// TIA Portal project "OPCUATST" (V15)

(* hardware
DEVICE "S71500/ET200MP station_1"  S7-1500 station
   slot 0: "导轨_0"  Rack  6ES7 590-1***0-0AA0
   slot 1: "PLC_1"  CPU 1515-2 PN  6ES7 515-2AM01-0AB0  V2.5
      slot 3: "CPU 显示_1"  6ES7591-1BA00-0AA0
*)

// ===== PLC "PLC_1"  CPU 1515-2 PN =====

VAR_GLOBAL   // PLC tag table "默认变量表"
   "OPCUATESTBOOL" AT %M0.0 : Bool;
   "OPCUATESTMW" AT %MW1 : Word;
   "OPCUATESTMD" AT %MD4 : DWord;
END_VAR

DATA_BLOCK "DataStatic"   // DB2
{ S7_Optimized_Access := 'TRUE' }
VERSION : 0.1
   VAR
      myBool : Bool := true;
      myByte : Byte := 16#AB;
      myWord : Word := 16#CDEF;
      myDword : DWord := 16#1234567F;
      myInt : Int := 42;
      myUInt : UInt := 65535;
      myString : String := 'Hello World';
      myReal : Real := 9.81;
      myArrayByte : Array[0..127] of Byte;
      myArrayInt : Array[0..127] of Int;
      myArrayUInt : Array[0..127] of UInt;
      myArrayLInt : Array[0..127] of LInt;
      myArrayReal : Array[0..127] of Real;
      myArrayLReal : Array[0..127] of LReal;
      myArrayBool : Array[0..127] of Bool;
   END_VAR
BEGIN
   myArrayByte[0] := 1;
   myArrayByte[1] := 2;
   myArrayByte[2] := 3;
   myArrayByte[3] := 4;
   myArrayByte[4] := 5;
   myArrayByte[5] := 6;
   myArrayByte[6] := 7;
   myArrayByte[7] := 8;
   myArrayByte[8] := 9;
   myArrayByte[9] := 10;
   myArrayByte[10] := 11;
   myArrayByte[11] := 12;
   myArrayByte[12] := 13;
   myArrayByte[13] := 14;
   myArrayByte[14] := 15;
   myArrayByte[15] := 16;
   myArrayByte[16] := 17;
   myArrayByte[17] := 18;
   myArrayByte[18] := 19;
   myArrayByte[19] := 20;
   myArrayByte[20] := 21;
   myArrayByte[21] := 22;
   myArrayByte[22] := 23;
   myArrayByte[23] := 24;
   myArrayByte[24] := 25;
   myArrayByte[25] := 26;
   myArrayByte[26] := 27;
   myArrayByte[27] := 28;
   myArrayByte[28] := 29;
   myArrayByte[29] := 30;
   myArrayByte[30] := 31;
   myArrayByte[31] := 32;
   myArrayByte[32] := 33;
   myArrayByte[33] := 34;
   myArrayByte[34] := 35;
   myArrayByte[35] := 36;
   myArrayByte[36] := 37;
   myArrayByte[37] := 38;
   myArrayByte[38] := 39;
   myArrayByte[39] := 40;
   myArrayByte[40] := 41;
   myArrayByte[41] := 42;
   myArrayByte[42] := 43;
   myArrayByte[43] := 44;
   myArrayByte[44] := 45;
   myArrayByte[45] := 46;
   myArrayByte[46] := 47;
   myArrayByte[47] := 48;
   myArrayByte[48] := 49;
   myArrayByte[49] := 50;
   myArrayByte[50] := 51;
   myArrayByte[51] := 52;
   myArrayByte[52] := 53;
   myArrayByte[53] := 54;
   myArrayByte[54] := 55;
   myArrayByte[55] := 56;
   myArrayByte[56] := 57;
   myArrayByte[57] := 58;
   myArrayByte[58] := 59;
   myArrayByte[59] := 60;
   myArrayByte[60] := 61;
   myArrayByte[61] := 62;
   myArrayByte[62] := 63;
   myArrayByte[63] := 64;
   myArrayByte[64] := 65;
   myArrayByte[65] := 66;
   myArrayByte[66] := 67;
   myArrayByte[67] := 68;
   myArrayByte[68] := 69;
   myArrayByte[69] := 70;
   myArrayByte[70] := 71;
   myArrayByte[71] := 72;
   myArrayByte[72] := 73;
   myArrayByte[73] := 74;
   myArrayByte[74] := 75;
   myArrayByte[75] := 76;
   myArrayByte[76] := 77;
   myArrayByte[77] := 78;
   myArrayByte[78] := 79;
   myArrayByte[79] := 80;
   myArrayByte[80] := 81;
   myArrayByte[81] := 82;
   myArrayByte[82] := 83;
   myArrayByte[83] := 84;
   myArrayByte[84] := 85;
   myArrayByte[85] := 86;
   myArrayByte[86] := 87;
   myArrayByte[87] := 88;
   myArrayByte[88] := 89;
   myArrayByte[89] := 90;
   myArrayByte[90] := 91;
   myArrayByte[91] := 92;
   myArrayByte[92] := 93;
   myArrayByte[93] := 94;
   myArrayByte[94] := 95;
   myArrayByte[95] := 96;
   myArrayByte[96] := 97;
   myArrayByte[97] := 98;
   myArrayByte[98] := 99;
   myArrayByte[99] := 100;
   myArrayByte[100] := 101;
   myArrayByte[101] := 102;
   myArrayByte[102] := 103;
   myArrayByte[103] := 104;
   myArrayByte[104] := 105;
   myArrayByte[105] := 106;
   myArrayByte[106] := 107;
   myArrayByte[107] := 108;
   myArrayByte[108] := 109;
   myArrayByte[109] := 110;
   myArrayByte[110] := 111;
   myArrayByte[111] := 112;
   myArrayByte[112] := 113;
   myArrayByte[113] := 114;
   myArrayByte[114] := 115;
   myArrayByte[115] := 116;
   myArrayByte[116] := 117;
   myArrayByte[117] := 118;
   myArrayByte[118] := 119;
   myArrayByte[119] := 120;
   myArrayByte[120] := 121;
   myArrayByte[121] := 122;
   myArrayByte[122] := 123;
   myArrayByte[123] := 124;
   myArrayByte[124] := 125;
   myArrayByte[125] := 126;
   myArrayByte[126] := 127;
   myArrayByte[127] := 128;
   myArrayInt[0] := 1;
   myArrayInt[1] := 2;
   myArrayInt[2] := 3;
   myArrayInt[3] := 4;
   myArrayInt[4] := 5;
   myArrayInt[5] := 6;
   myArrayInt[6] := 7;
   myArrayInt[7] := 8;
   myArrayInt[8] := 9;
   myArrayInt[9] := 10;
   myArrayInt[10] := 11;
   myArrayInt[11] := 12;
   myArrayInt[12] := 13;
   myArrayInt[13] := 14;
   myArrayInt[14] := 15;
   myArrayInt[15] := 16;
   myArrayInt[16] := 17;
   myArrayInt[17] := 18;
   myArrayInt[18] := 19;
   myArrayInt[19] := 20;
   myArrayInt[20] := 21;
   myArrayInt[21] := 22;
   myArrayInt[22] := 23;
   myArrayInt[23] := 24;
   myArrayInt[24] := 25;
   myArrayInt[25] := 26;
   myArrayInt[26] := 27;
   myArrayInt[27] := 28;
   myArrayInt[28] := 29;
   myArrayInt[29] := 30;
   myArrayInt[30] := 31;
   myArrayInt[31] := 32;
   myArrayInt[32] := 33;
   myArrayInt[33] := 34;
   myArrayInt[34] := 35;
   myArrayInt[35] := 36;
   myArrayInt[36] := 37;
   myArrayInt[37] := 38;
   myArrayInt[38] := 39;
   myArrayInt[39] := 40;
   myArrayInt[40] := 41;
   myArrayInt[41] := 42;
   myArrayInt[42] := 43;
   myArrayInt[43] := 44;
   myArrayInt[44] := 45;
   myArrayInt[45] := 46;
   myArrayInt[46] := 47;
   myArrayInt[47] := 48;
   myArrayInt[48] := 49;
   myArrayInt[49] := 50;
   myArrayInt[50] := 51;
   myArrayInt[51] := 52;
   myArrayInt[52] := 53;
   myArrayInt[53] := 54;
   myArrayInt[54] := 55;
   myArrayInt[55] := 56;
   myArrayInt[56] := 57;
   myArrayInt[57] := 58;
   myArrayInt[58] := 59;
   myArrayInt[59] := 60;
   myArrayInt[60] := 61;
   myArrayInt[61] := 62;
   myArrayInt[62] := 63;
   myArrayInt[63] := 64;
   myArrayInt[64] := 65;
   myArrayInt[65] := 66;
   myArrayInt[66] := 67;
   myArrayInt[67] := 68;
   myArrayInt[68] := 69;
   myArrayInt[69] := 70;
   myArrayInt[70] := 71;
   myArrayInt[71] := 72;
   myArrayInt[72] := 73;
   myArrayInt[73] := 74;
   myArrayInt[74] := 75;
   myArrayInt[75] := 76;
   myArrayInt[76] := 77;
   myArrayInt[77] := 78;
   myArrayInt[78] := 79;
   myArrayInt[79] := 80;
   myArrayInt[80] := 81;
   myArrayInt[81] := 82;
   myArrayInt[82] := 83;
   myArrayInt[83] := 84;
   myArrayInt[84] := 85;
   myArrayInt[85] := 86;
   myArrayInt[86] := 87;
   myArrayInt[87] := 88;
   myArrayInt[88] := 89;
   myArrayInt[89] := 90;
   myArrayInt[90] := 91;
   myArrayInt[91] := 92;
   myArrayInt[92] := 93;
   myArrayInt[93] := 94;
   myArrayInt[94] := 95;
   myArrayInt[95] := 96;
   myArrayInt[96] := 97;
   myArrayInt[97] := 98;
   myArrayInt[98] := 99;
   myArrayInt[99] := 100;
   myArrayInt[100] := 101;
   myArrayInt[101] := 102;
   myArrayInt[102] := 103;
   myArrayInt[103] := 104;
   myArrayInt[104] := 105;
   myArrayInt[105] := 106;
   myArrayInt[106] := 107;
   myArrayInt[107] := 108;
   myArrayInt[108] := 109;
   myArrayInt[109] := 110;
   myArrayInt[110] := 111;
   myArrayInt[111] := 112;
   myArrayInt[112] := 113;
   myArrayInt[113] := 114;
   myArrayInt[114] := 115;
   myArrayInt[115] := 116;
   myArrayInt[116] := 117;
   myArrayInt[117] := 118;
   myArrayInt[118] := 119;
   myArrayInt[119] := 120;
   myArrayInt[120] := 121;
   myArrayInt[121] := 122;
   myArrayInt[122] := 123;
   myArrayInt[123] := 124;
   myArrayInt[124] := 125;
   myArrayInt[125] := 126;
   myArrayInt[126] := 127;
   myArrayInt[127] := 128;
   myArrayUInt[0] := 1;
   myArrayUInt[1] := 2;
   myArrayUInt[2] := 3;
   myArrayUInt[3] := 4;
   myArrayUInt[4] := 5;
   myArrayUInt[5] := 6;
   myArrayUInt[6] := 7;
   myArrayUInt[7] := 8;
   myArrayUInt[8] := 9;
   myArrayUInt[9] := 10;
   myArrayUInt[10] := 11;
   myArrayUInt[11] := 12;
   myArrayUInt[12] := 13;
   myArrayUInt[13] := 14;
   myArrayUInt[14] := 15;
   myArrayUInt[15] := 16;
   myArrayUInt[16] := 17;
   myArrayUInt[17] := 18;
   myArrayUInt[18] := 19;
   myArrayUInt[19] := 20;
   myArrayUInt[20] := 21;
   myArrayUInt[21] := 22;
   myArrayUInt[22] := 23;
   myArrayUInt[23] := 24;
   myArrayUInt[24] := 25;
   myArrayUInt[25] := 26;
   myArrayUInt[26] := 27;
   myArrayUInt[27] := 28;
   myArrayUInt[28] := 29;
   myArrayUInt[29] := 30;
   myArrayUInt[30] := 31;
   myArrayUInt[31] := 32;
   myArrayUInt[32] := 33;
   myArrayUInt[33] := 34;
   myArrayUInt[34] := 35;
   myArrayUInt[35] := 36;
   myArrayUInt[36] := 37;
   myArrayUInt[37] := 38;
   myArrayUInt[38] := 39;
   myArrayUInt[39] := 40;
   myArrayUInt[40] := 41;
   myArrayUInt[41] := 42;
   myArrayUInt[42] := 43;
   myArrayUInt[43] := 44;
   myArrayUInt[44] := 45;
   myArrayUInt[45] := 46;
   myArrayUInt[46] := 47;
   myArrayUInt[47] := 48;
   myArrayUInt[48] := 49;
   myArrayUInt[49] := 50;
   myArrayUInt[50] := 51;
   myArrayUInt[51] := 52;
   myArrayUInt[52] := 53;
   myArrayUInt[53] := 54;
   myArrayUInt[54] := 55;
   myArrayUInt[55] := 56;
   myArrayUInt[56] := 57;
   myArrayUInt[57] := 58;
   myArrayUInt[58] := 59;
   myArrayUInt[59] := 60;
   myArrayUInt[60] := 61;
   myArrayUInt[61] := 62;
   myArrayUInt[62] := 63;
   myArrayUInt[63] := 64;
   myArrayUInt[64] := 65;
   myArrayUInt[65] := 66;
   myArrayUInt[66] := 67;
   myArrayUInt[67] := 68;
   myArrayUInt[68] := 69;
   myArrayUInt[69] := 70;
   myArrayUInt[70] := 71;
   myArrayUInt[71] := 72;
   myArrayUInt[72] := 73;
   myArrayUInt[73] := 74;
   myArrayUInt[74] := 75;
   myArrayUInt[75] := 76;
   myArrayUInt[76] := 77;
   myArrayUInt[77] := 78;
   myArrayUInt[78] := 79;
   myArrayUInt[79] := 80;
   myArrayUInt[80] := 81;
   myArrayUInt[81] := 82;
   myArrayUInt[82] := 83;
   myArrayUInt[83] := 84;
   myArrayUInt[84] := 85;
   myArrayUInt[85] := 86;
   myArrayUInt[86] := 87;
   myArrayUInt[87] := 88;
   myArrayUInt[88] := 89;
   myArrayUInt[89] := 90;
   myArrayUInt[90] := 91;
   myArrayUInt[91] := 92;
   myArrayUInt[92] := 93;
   myArrayUInt[93] := 94;
   myArrayUInt[94] := 95;
   myArrayUInt[95] := 96;
   myArrayUInt[96] := 97;
   myArrayUInt[97] := 98;
   myArrayUInt[98] := 99;
   myArrayUInt[99] := 100;
   myArrayUInt[100] := 101;
   myArrayUInt[101] := 102;
   myArrayUInt[102] := 103;
   myArrayUInt[103] := 104;
   myArrayUInt[104] := 105;
   myArrayUInt[105] := 106;
   myArrayUInt[106] := 107;
   myArrayUInt[107] := 108;
   myArrayUInt[108] := 109;
   myArrayUInt[109] := 110;
   myArrayUInt[110] := 111;
   myArrayUInt[111] := 112;
   myArrayUInt[112] := 113;
   myArrayUInt[113] := 114;
   myArrayUInt[114] := 115;
   myArrayUInt[115] := 116;
   myArrayUInt[116] := 117;
   myArrayUInt[117] := 118;
   myArrayUInt[118] := 119;
   myArrayUInt[119] := 120;
   myArrayUInt[120] := 121;
   myArrayUInt[121] := 122;
   myArrayUInt[122] := 123;
   myArrayUInt[123] := 124;
   myArrayUInt[124] := 125;
   myArrayUInt[125] := 126;
   myArrayUInt[126] := 127;
   myArrayUInt[127] := 128;
   myArrayLInt[0] := 1;
   myArrayLInt[1] := 2;
   myArrayLInt[2] := 3;
   myArrayLInt[3] := 4;
   myArrayLInt[4] := 5;
   myArrayLInt[5] := 6;
   myArrayLInt[6] := 7;
   myArrayLInt[7] := 8;
   myArrayLInt[8] := 9;
   myArrayLInt[9] := 10;
   myArrayLInt[10] := 11;
   myArrayLInt[11] := 12;
   myArrayLInt[12] := 13;
   myArrayLInt[13] := 14;
   myArrayLInt[14] := 15;
   myArrayLInt[15] := 16;
   myArrayLInt[16] := 17;
   myArrayLInt[17] := 18;
   myArrayLInt[18] := 19;
   myArrayLInt[19] := 20;
   myArrayLInt[20] := 21;
   myArrayLInt[21] := 22;
   myArrayLInt[22] := 23;
   myArrayLInt[23] := 24;
   myArrayLInt[24] := 25;
   myArrayLInt[25] := 26;
   myArrayLInt[26] := 27;
   myArrayLInt[27] := 28;
   myArrayLInt[28] := 29;
   myArrayLInt[29] := 30;
   myArrayLInt[30] := 31;
   myArrayLInt[31] := 32;
   myArrayLInt[32] := 33;
   myArrayLInt[33] := 34;
   myArrayLInt[34] := 35;
   myArrayLInt[35] := 36;
   myArrayLInt[36] := 37;
   myArrayLInt[37] := 38;
   myArrayLInt[38] := 39;
   myArrayLInt[39] := 40;
   myArrayLInt[40] := 41;
   myArrayLInt[41] := 42;
   myArrayLInt[42] := 43;
   myArrayLInt[43] := 44;
   myArrayLInt[44] := 45;
   myArrayLInt[45] := 46;
   myArrayLInt[46] := 47;
   myArrayLInt[47] := 48;
   myArrayLInt[48] := 49;
   myArrayLInt[49] := 50;
   myArrayLInt[50] := 51;
   myArrayLInt[51] := 52;
   myArrayLInt[52] := 53;
   myArrayLInt[53] := 54;
   myArrayLInt[54] := 55;
   myArrayLInt[55] := 56;
   myArrayLInt[56] := 57;
   myArrayLInt[57] := 58;
   myArrayLInt[58] := 59;
   myArrayLInt[59] := 60;
   myArrayLInt[60] := 61;
   myArrayLInt[61] := 62;
   myArrayLInt[62] := 63;
   myArrayLInt[63] := 64;
   myArrayLInt[64] := 65;
   myArrayLInt[65] := 66;
   myArrayLInt[66] := 67;
   myArrayLInt[67] := 68;
   myArrayLInt[68] := 69;
   myArrayLInt[69] := 70;
   myArrayLInt[70] := 71;
   myArrayLInt[71] := 72;
   myArrayLInt[72] := 73;
   myArrayLInt[73] := 74;
   myArrayLInt[74] := 75;
   myArrayLInt[75] := 76;
   myArrayLInt[76] := 77;
   myArrayLInt[77] := 78;
   myArrayLInt[78] := 79;
   myArrayLInt[79] := 80;
   myArrayLInt[80] := 81;
   myArrayLInt[81] := 82;
   myArrayLInt[82] := 83;
   myArrayLInt[83] := 84;
   myArrayLInt[84] := 85;
   myArrayLInt[85] := 86;
   myArrayLInt[86] := 87;
   myArrayLInt[87] := 88;
   myArrayLInt[88] := 89;
   myArrayLInt[89] := 90;
   myArrayLInt[90] := 91;
   myArrayLInt[91] := 92;
   myArrayLInt[92] := 93;
   myArrayLInt[93] := 94;
   myArrayLInt[94] := 95;
   myArrayLInt[95] := 96;
   myArrayLInt[96] := 97;
   myArrayLInt[97] := 98;
   myArrayLInt[98] := 99;
   myArrayLInt[99] := 100;
   myArrayLInt[100] := 101;
   myArrayLInt[101] := 102;
   myArrayLInt[102] := 103;
   myArrayLInt[103] := 104;
   myArrayLInt[104] := 105;
   myArrayLInt[105] := 106;
   myArrayLInt[106] := 107;
   myArrayLInt[107] := 108;
   myArrayLInt[108] := 109;
   myArrayLInt[109] := 110;
   myArrayLInt[110] := 111;
   myArrayLInt[111] := 112;
   myArrayLInt[112] := 113;
   myArrayLInt[113] := 114;
   myArrayLInt[114] := 115;
   myArrayLInt[115] := 116;
   myArrayLInt[116] := 117;
   myArrayLInt[117] := 118;
   myArrayLInt[118] := 119;
   myArrayLInt[119] := 120;
   myArrayLInt[120] := 121;
   myArrayLInt[121] := 122;
   myArrayLInt[122] := 123;
   myArrayLInt[123] := 124;
   myArrayLInt[124] := 125;
   myArrayLInt[125] := 126;
   myArrayLInt[126] := 127;
   myArrayLInt[127] := 128;
   myArrayReal[0] := 1.1;
   myArrayReal[1] := 2.0;
   myArrayReal[2] := 3.0;
   myArrayReal[3] := 4.456;
   myArrayReal[4] := 5.0;
   myArrayReal[5] := 6.0;
   myArrayReal[6] := 7.0;
   myArrayReal[7] := 8.0;
   myArrayReal[8] := 9.0;
   myArrayReal[9] := 10.0;
   myArrayReal[10] := 11.0;
   myArrayReal[11] := 12.0;
   myArrayReal[12] := 13.0;
   myArrayReal[13] := 14.0;
   myArrayReal[14] := 15.0;
   myArrayReal[15] := 16.0;
   myArrayReal[16] := 17.0;
   myArrayReal[17] := 18.0;
   myArrayReal[18] := 19.0;
   myArrayReal[19] := 20.0;
   myArrayReal[20] := 21.0;
   myArrayReal[21] := 22.0;
   myArrayReal[22] := 23.0;
   myArrayReal[23] := 24.0;
   myArrayReal[24] := 25.0;
   myArrayReal[25] := 26.0;
   myArrayReal[26] := 27.0;
   myArrayReal[27] := 28.0;
   myArrayReal[28] := 29.0;
   myArrayReal[29] := 30.0;
   myArrayReal[30] := 31.0;
   myArrayReal[31] := 32.0;
   myArrayReal[32] := 33.0;
   myArrayReal[33] := 34.0;
   myArrayReal[34] := 35.0;
   myArrayReal[35] := 36.0;
   myArrayReal[36] := 37.0;
   myArrayReal[37] := 38.0;
   myArrayReal[38] := 39.0;
   myArrayReal[39] := 40.0;
   myArrayReal[40] := 41.0;
   myArrayReal[41] := 42.0;
   myArrayReal[42] := 43.0;
   myArrayReal[43] := 44.0;
   myArrayReal[44] := 45.0;
   myArrayReal[45] := 46.0;
   myArrayReal[46] := 47.0;
   myArrayReal[47] := 48.0;
   myArrayReal[48] := 49.0;
   myArrayReal[49] := 50.0;
   myArrayReal[50] := 51.0;
   myArrayReal[51] := 52.0;
   myArrayReal[52] := 53.0;
   myArrayReal[53] := 54.0;
   myArrayReal[54] := 55.0;
   myArrayReal[55] := 56.0;
   myArrayReal[56] := 57.0;
   myArrayReal[57] := 58.0;
   myArrayReal[58] := 59.0;
   myArrayReal[59] := 60.0;
   myArrayReal[60] := 61.0;
   myArrayReal[61] := 62.0;
   myArrayReal[62] := 63.0;
   myArrayReal[63] := 64.0;
   myArrayReal[64] := 65.0;
   myArrayReal[65] := 66.0;
   myArrayReal[66] := 67.0;
   myArrayReal[67] := 68.0;
   myArrayReal[68] := 69.0;
   myArrayReal[69] := 70.0;
   myArrayReal[70] := 71.0;
   myArrayReal[71] := 72.0;
   myArrayReal[72] := 73.0;
   myArrayReal[73] := 74.0;
   myArrayReal[74] := 75.0;
   myArrayReal[75] := 76.0;
   myArrayReal[76] := 77.0;
   myArrayReal[77] := 78.0;
   myArrayReal[78] := 79.0;
   myArrayReal[79] := 80.0;
   myArrayReal[80] := 81.0;
   myArrayReal[81] := 82.0;
   myArrayReal[82] := 83.0;
   myArrayReal[83] := 84.0;
   myArrayReal[84] := 85.0;
   myArrayReal[85] := 86.0;
   myArrayReal[86] := 87.0;
   myArrayReal[87] := 88.0;
   myArrayReal[88] := 89.0;
   myArrayReal[89] := 90.0;
   myArrayReal[90] := 91.0;
   myArrayReal[91] := 92.0;
   myArrayReal[92] := 93.0;
   myArrayReal[93] := 94.0;
   myArrayReal[94] := 95.0;
   myArrayReal[95] := 96.0;
   myArrayReal[96] := 97.0;
   myArrayReal[97] := 98.0;
   myArrayReal[98] := 99.0;
   myArrayReal[99] := 100.0;
   myArrayReal[100] := 101.0;
   myArrayReal[101] := 102.0;
   myArrayReal[102] := 103.0;
   myArrayReal[103] := 104.0;
   myArrayReal[104] := 105.0;
   myArrayReal[105] := 106.0;
   myArrayReal[106] := 107.0;
   myArrayReal[107] := 108.0;
   myArrayReal[108] := 109.0;
   myArrayReal[109] := 110.0;
   myArrayReal[110] := 111.0;
   myArrayReal[111] := 112.0;
   myArrayReal[112] := 113.0;
   myArrayReal[113] := 114.0;
   myArrayReal[114] := 115.0;
   myArrayReal[115] := 116.0;
   myArrayReal[116] := 117.0;
   myArrayReal[117] := 118.0;
   myArrayReal[118] := 119.0;
   myArrayReal[119] := 120.0;
   myArrayReal[120] := 121.0;
   myArrayReal[121] := 122.0;
   myArrayReal[122] := 123.0;
   myArrayReal[123] := 124.0;
   myArrayReal[124] := 125.0;
   myArrayReal[125] := 126.0;
   myArrayReal[126] := 127.0;
   myArrayReal[127] := 128.0;
   myArrayLReal[0] := 1.0;
   myArrayLReal[1] := 2.0;
   myArrayLReal[2] := 3.0;
   myArrayLReal[3] := 4.0;
   myArrayLReal[4] := 5.0;
   myArrayLReal[5] := 6.0;
   myArrayLReal[6] := 7.0;
   myArrayLReal[7] := 8.0;
   myArrayLReal[8] := 9.0;
   myArrayLReal[9] := 10.0;
   myArrayLReal[10] := 11.0;
   myArrayLReal[11] := 12.0;
   myArrayLReal[12] := 13.0;
   myArrayLReal[13] := 14.0;
   myArrayLReal[14] := 15.0;
   myArrayLReal[15] := 16.0;
   myArrayLReal[16] := 17.0;
   myArrayLReal[17] := 18.0;
   myArrayLReal[18] := 19.0;
   myArrayLReal[19] := 20.0;
   myArrayLReal[20] := 21.0;
   myArrayLReal[21] := 22.0;
   myArrayLReal[22] := 23.0;
   myArrayLReal[23] := 24.0;
   myArrayLReal[24] := 25.0;
   myArrayLReal[25] := 26.0;
   myArrayLReal[26] := 27.0;
   myArrayLReal[27] := 28.0;
   myArrayLReal[28] := 29.0;
   myArrayLReal[29] := 30.0;
   myArrayLReal[30] := 31.0;
   myArrayLReal[31] := 32.0;
   myArrayLReal[32] := 33.0;
   myArrayLReal[33] := 34.0;
   myArrayLReal[34] := 35.0;
   myArrayLReal[35] := 36.0;
   myArrayLReal[36] := 37.0;
   myArrayLReal[37] := 38.0;
   myArrayLReal[38] := 39.0;
   myArrayLReal[39] := 40.0;
   myArrayLReal[40] := 41.0;
   myArrayLReal[41] := 42.0;
   myArrayLReal[42] := 43.0;
   myArrayLReal[43] := 44.0;
   myArrayLReal[44] := 45.0;
   myArrayLReal[45] := 46.0;
   myArrayLReal[46] := 47.0;
   myArrayLReal[47] := 48.0;
   myArrayLReal[48] := 49.0;
   myArrayLReal[49] := 50.0;
   myArrayLReal[50] := 51.0;
   myArrayLReal[51] := 52.0;
   myArrayLReal[52] := 53.0;
   myArrayLReal[53] := 54.0;
   myArrayLReal[54] := 55.0;
   myArrayLReal[55] := 56.0;
   myArrayLReal[56] := 57.0;
   myArrayLReal[57] := 58.0;
   myArrayLReal[58] := 59.0;
   myArrayLReal[59] := 60.0;
   myArrayLReal[60] := 61.0;
   myArrayLReal[61] := 62.0;
   myArrayLReal[62] := 63.0;
   myArrayLReal[63] := 64.0;
   myArrayLReal[64] := 65.0;
   myArrayLReal[65] := 66.0;
   myArrayLReal[66] := 67.0;
   myArrayLReal[67] := 68.0;
   myArrayLReal[68] := 69.0;
   myArrayLReal[69] := 70.0;
   myArrayLReal[70] := 71.0;
   myArrayLReal[71] := 72.0;
   myArrayLReal[72] := 73.0;
   myArrayLReal[73] := 74.0;
   myArrayLReal[74] := 75.0;
   myArrayLReal[75] := 76.0;
   myArrayLReal[76] := 77.0;
   myArrayLReal[77] := 78.0;
   myArrayLReal[78] := 79.0;
   myArrayLReal[79] := 80.0;
   myArrayLReal[80] := 81.0;
   myArrayLReal[81] := 82.0;
   myArrayLReal[82] := 83.0;
   myArrayLReal[83] := 84.0;
   myArrayLReal[84] := 85.0;
   myArrayLReal[85] := 86.0;
   myArrayLReal[86] := 87.0;
   myArrayLReal[87] := 88.0;
   myArrayLReal[88] := 89.0;
   myArrayLReal[89] := 90.0;
   myArrayLReal[90] := 91.0;
   myArrayLReal[91] := 92.0;
   myArrayLReal[92] := 93.0;
   myArrayLReal[93] := 94.0;
   myArrayLReal[94] := 95.0;
   myArrayLReal[95] := 96.0;
   myArrayLReal[96] := 97.0;
   myArrayLReal[97] := 98.0;
   myArrayLReal[98] := 99.0;
   myArrayLReal[99] := 100.0;
   myArrayLReal[100] := 101.0;
   myArrayLReal[101] := 102.0;
   myArrayLReal[102] := 103.0;
   myArrayLReal[103] := 104.0;
   myArrayLReal[104] := 105.0;
   myArrayLReal[105] := 106.0;
   myArrayLReal[106] := 107.0;
   myArrayLReal[107] := 108.0;
   myArrayLReal[108] := 109.0;
   myArrayLReal[109] := 110.0;
   myArrayLReal[110] := 111.0;
   myArrayLReal[111] := 112.0;
   myArrayLReal[112] := 113.0;
   myArrayLReal[113] := 114.0;
   myArrayLReal[114] := 115.0;
   myArrayLReal[115] := 116.0;
   myArrayLReal[116] := 117.0;
   myArrayLReal[117] := 118.0;
   myArrayLReal[118] := 119.0;
   myArrayLReal[119] := 120.0;
   myArrayLReal[120] := 121.0;
   myArrayLReal[121] := 122.0;
   myArrayLReal[122] := 123.0;
   myArrayLReal[123] := 124.0;
   myArrayLReal[124] := 125.0;
   myArrayLReal[125] := 126.0;
   myArrayLReal[126] := 127.0;
   myArrayLReal[127] := 128.0;
   myArrayBool[0] := true;
   myArrayBool[1] := false;
   myArrayBool[2] := true;
   myArrayBool[3] := false;
   myArrayBool[4] := true;
   myArrayBool[5] := false;
   myArrayBool[6] := true;
   myArrayBool[7] := false;
   myArrayBool[8] := true;
   myArrayBool[9] := false;
   myArrayBool[10] := true;
   myArrayBool[11] := false;
   myArrayBool[12] := true;
   myArrayBool[13] := false;
   myArrayBool[14] := true;
   myArrayBool[15] := false;
   myArrayBool[16] := true;
   myArrayBool[17] := false;
   myArrayBool[18] := true;
   myArrayBool[19] := false;
   myArrayBool[20] := true;
   myArrayBool[21] := true;
   myArrayBool[22] := false;
   myArrayBool[23] := true;
   myArrayBool[24] := false;
   myArrayBool[25] := true;
   myArrayBool[26] := false;
   myArrayBool[27] := true;
   myArrayBool[28] := false;
   myArrayBool[29] := true;
   myArrayBool[30] := false;
   myArrayBool[31] := true;
   myArrayBool[32] := false;
   myArrayBool[33] := true;
   myArrayBool[34] := false;
   myArrayBool[35] := true;
   myArrayBool[36] := false;
   myArrayBool[37] := true;
   myArrayBool[38] := false;
   myArrayBool[39] := true;
   myArrayBool[40] := false;
   myArrayBool[41] := true;
   myArrayBool[42] := true;
   myArrayBool[43] := false;
   myArrayBool[44] := true;
   myArrayBool[45] := false;
   myArrayBool[46] := true;
   myArrayBool[47] := false;
   myArrayBool[48] := true;
   myArrayBool[49] := false;
   myArrayBool[50] := true;
   myArrayBool[51] := false;
   myArrayBool[52] := true;
   myArrayBool[53] := false;
   myArrayBool[54] := true;
   myArrayBool[55] := false;
   myArrayBool[56] := true;
   myArrayBool[57] := false;
   myArrayBool[58] := true;
   myArrayBool[59] := false;
   myArrayBool[60] := true;
   myArrayBool[61] := false;
   myArrayBool[62] := true;
   myArrayBool[63] := true;
   myArrayBool[64] := false;
   myArrayBool[65] := true;
   myArrayBool[66] := false;
   myArrayBool[67] := true;
   myArrayBool[68] := false;
   myArrayBool[69] := true;
   myArrayBool[70] := false;
   myArrayBool[71] := true;
   myArrayBool[72] := false;
   myArrayBool[73] := true;
   myArrayBool[74] := false;
   myArrayBool[75] := true;
   myArrayBool[76] := false;
   myArrayBool[77] := true;
   myArrayBool[78] := false;
   myArrayBool[79] := true;
   myArrayBool[80] := false;
   myArrayBool[81] := true;
   myArrayBool[82] := false;
   myArrayBool[83] := true;
   myArrayBool[84] := true;
   myArrayBool[85] := false;
   myArrayBool[86] := true;
   myArrayBool[87] := false;
   myArrayBool[88] := true;
   myArrayBool[89] := false;
   myArrayBool[90] := true;
   myArrayBool[91] := false;
   myArrayBool[92] := true;
   myArrayBool[93] := false;
   myArrayBool[94] := true;
   myArrayBool[95] := false;
   myArrayBool[96] := true;
   myArrayBool[97] := false;
   myArrayBool[98] := true;
   myArrayBool[99] := false;
   myArrayBool[100] := true;
   myArrayBool[101] := false;
   myArrayBool[102] := true;
   myArrayBool[103] := false;
   myArrayBool[104] := true;
   myArrayBool[105] := true;
   myArrayBool[106] := false;
   myArrayBool[107] := true;
   myArrayBool[108] := false;
   myArrayBool[109] := true;
   myArrayBool[110] := false;
   myArrayBool[111] := true;
   myArrayBool[112] := false;
   myArrayBool[113] := true;
   myArrayBool[114] := false;
   myArrayBool[115] := true;
   myArrayBool[116] := false;
   myArrayBool[117] := true;
   myArrayBool[118] := false;
   myArrayBool[119] := true;
   myArrayBool[120] := false;
   myArrayBool[121] := true;
   myArrayBool[122] := false;
   myArrayBool[123] := true;
   myArrayBool[124] := false;
   myArrayBool[125] := true;
   myArrayBool[126] := true;
   myArrayBool[127] := false;
END_DATA_BLOCK

DATA_BLOCK "State"   // DB100
{ S7_Optimized_Access := 'TRUE' }
VERSION : 0.1
   VAR RETAIN
      AC_X : Int;
      AC_Y : Int;
      ALIG_X : Int;
      ALIG_Y : Int;
      DC_X : Int;
      DC_Y : Int;
      PLC_Tag_P1 : Bool;
      PLC_Tag_P2 : Bool;
      PLC_Tag_P3 : Bool;
      PLC_Tag_P4 : Bool;
      PLC_Tag_P5 : Bool;
      PLC_Tag_P6 : Bool;
      HMI_Tag_P1_AL : Bool;
      HMI_Tag_P2_AL : Bool;
      HMI_Tag_P3_AL : Bool;
      HMI_Tag_P4_AL : Bool;
      HMI_Tag_P5_AL : Bool;
      HMI_Tag_P6_AL : Bool;
      PLC_Tag_V1 : Bool;
      PLC_Tag_V2 : Bool;
      PLC_Tag_V3 : Bool;
      PLC_Tag_V4 : Bool;
      PLC_Tag_V5 : Bool;
      PLC_Tag_V6 : Bool;
      PLC_Tag_V7 : Bool;
      HMI_Tag_V1_AL : Bool;
      HMI_Tag_V2_AL : Bool;
      HMI_Tag_V3_AL : Bool;
      HMI_Tag_V4_AL : Bool;
      HMI_Tag_V5_AL : Bool;
      HMI_Tag_V6_AL : Bool;
      HMI_Tag_V7_AL : Bool;
      HMI_Tag_VG1_AL : Bool;
      HMI_Tag_VG2_AL : Bool;
      HMI_Tag_VG3_AL : Bool;
      HMI_Tag_VG1 : Real;
      HMI_Tag_VG2 : Real;
      HMI_Tag_VG3 : Real;
      HMI_Tag_VG4 : Real;
      HV_MEASURE_VAL : Real;
      HV_SET_VAL : Real;
      IB_MEASURE_VAL : Real;
      IB_SET_VAL : Real;
      IF_MEASURE_VAL : Int;
      IF_SET_VAL : Int;
      IH_MEASURE_VAL : Real;
      IH_SET_VAL : Real;
      P2_WAU1001_ON_P : Real := 10000.0;
      P2_WAU1001_OFF_P : Real := 12000.0;
      SET_HV : Bool;
      SET_IB : Bool;
      SET_IF : Bool;
      SET_IH : Bool;
      DEFLECTION_WAVEFORM : Int;
      DEFLECTION_FREQUENCY : Int;
      COOLING_WATER_OK : Bool;
      MOL_START_VACUUM_P : Real;
      MOL_OFF_VACUUM_P : Real;
      DIFF_FRONT_VACUMM_OK : Real := 30.0;
      DIFF_FRONT_VACUMM_NOT_OK : Real := 50.0;
      COMPRESSED_AIR_OK : Bool;
      CHAMBER_LOW_VACUUM_P : Real;
      CHAMBER_LOW_VACUUM_NOTOK : Real;
      CHAMBER_VACUUM_OK : Bool;
      CHAMBER_VACUUM_OK_P : Real;
      CHAMBER_VACUUM_NOT_OK_P : Real;
      BEAM_UP_TON : Real;
      BEAM_DOWN_TON : Real;
      BEAM_SET_G : Real;
      BEAM_SET_O : Real;
      BEAM_SAMPLE_G : Real;
      BEAM_SAMPLE_O : Real;
      GENERATOR_OK : Bool;
      GENERATOR_OK_P : Real;
      GENERATOR_NOT_OK_P : Real;
      FILAMENT_HEAT_OK : Bool;
      FILAMENT_SET_G : Real;
      FILAMENT_SET_O : Real;
      FILAMENT_SAMPLE_G : Real;
      FILAMENT_SAMPLE_O : Real;
      CHAMBER_DOOR_CLOSE : Bool;
      FOCUS_SET_G : Real;
      FOCUS_SET_O : Real;
      FOCUS_SAMPLE_G : Real;
      FOCUS_SAMPLE_O : Real;
      HV_OK : Bool;
      HV_SET_G : Real;
      HV_SET_O : Real;
      HV_SAMPLE_G : Real;
      HV_SAMPLE_O : Real;
      Generator_evacuum_flag : Bool;
      Generator_vent_flag : Bool;
   END_VAR
BEGIN
END_DATA_BLOCK

ORGANIZATION_BLOCK "Main"   // OB1, LAD, ProgramCycle
TITLE = "Main Program Sweep (Cycle)"
{ S7_Optimized_Access := 'TRUE' }
VERSION : 0.1
   VAR_INPUT
      Initial_Call : Bool;   // Initial call of this OB
      Remanence : Bool;   // =True, if remanent data are available
   END_VAR
BEGIN
END_ORGANIZATION_BLOCK